// TIA Portal V19 export
DATA_BLOCK "A02_Carriage"   // DB159, Motion_DB
// stored: InstanceOfName TO_SynchronousAxis, OfSystemLibElement TO_SynchronousAxis, OfSystemLibVersion 8.0
TO_SynchronousAxis   // technology object, version 8.0
// stored: Connection Interface Actor, InputAddress 3264, OutputAddress 3264
// stored: Connection Interface Sensor[1], InputAddress 3264, OutputAddress 3264, SensorIndexInActorTelegram 1
// stored: Connection Interface Sensor[2], InputAddress 3264, OutputAddress 3264, SensorIndexInActorTelegram 2
// stored: ActualValueCoupling Ref A02_Rollformer, Type TO_PositioningAxis
   // // inherited from TO_PositioningAxis
   // // inherited from TO_SpeedAxis
   // // inherited from TO_Axis
   // // inherited from TO_Object
   // VAR
   //    Actor : TO_Struct_Actor;
   //    DynamicLimits : TO_Struct_DynamicLimits;
   //    DynamicDefaults : TO_Struct_DynamicDefaults;
   // END_VAR
   // VAR
   //    Sensor : Array[1..4] of TO_Struct_Sensor;
   //    Mechanics : TO_Struct_Mechanics;
   //    PositionLimits_HW : TO_Struct_PositionLimitsHW;
   //    Homing : TO_Struct_Homing;
   //    PositionControl : TO_Struct_PositionControl;
   //    DynamicAxisModel : TO_Struct_DynamicAxisModel;
   //    FollowingError : TO_Struct_FollowingError;
   //    StandstillSignal : TO_Struct_StandstillSignal;
   // END_VAR
   // VAR
   //    StatusSynchronizedMotion { ExternalWritable := 'False'; S7_SetPoint := 'True'} : TO_Struct_StatusSynchronizedMotion;
   // END_VAR
BEGIN
   Actor.DataAdaption := 1;
   Actor.Interface.AddressIn.RID := 16#208072c;
   Actor.Interface.AddressIn.AREA := 16#81;
   Actor.Interface.AddressIn.OFFSET := 3264;
   Actor.Interface.AddressOut.RID := 16#208072d;
   Actor.Interface.AddressOut.AREA := 16#82;
   Actor.Interface.AddressOut.OFFSET := 3264;
   Actor.DriveParameter.ReferenceSpeed := 2000.0;
   Actor.DriveParameter.MaxSpeed := 4046.462;
   Actor.DriveParameter.ReferenceTorque := 168.27;
   DynamicLimits.MaxVelocity := 50000.0;
   DynamicLimits.Velocity := 50000.0;
   DynamicLimits.MaxAcceleration := 5000.0;
   DynamicLimits.MaxDeceleration := 5000.0;
   DynamicLimits.MaxJerk := 99999.9999999997;
   DynamicDefaults.Velocity := 6000.0;
   DynamicDefaults.EmergencyDeceleration := 5000.0;
   Sensor[2].Existent := true;
   Sensor[1]."Type" := 2;
   Sensor[2].System := 0;
   Sensor[1..2].DataAdaption := 1;
   Sensor[1].ActualVelocityMode := 1;
   Sensor[1..2].Interface.AddressIn.RID := 16#208072c;
   Sensor[1..2].Interface.AddressIn.AREA := 16#81;
   Sensor[1..2].Interface.AddressIn.OFFSET := 3264;
   Sensor[1..2].Interface.AddressOut.RID := 16#208072d;
   Sensor[1..2].Interface.AddressOut.AREA := 16#82;
   Sensor[1..2].Interface.AddressOut.OFFSET := 3264;
   Sensor[2].Interface.Number := 2;
   Sensor[2].Parameter.Resolution := 0.004;
   Sensor[1].Parameter.DeterminableRevolutions := 4096;
   Sensor[1].Parameter.ReferenceSpeed := 2000.0;
   Mechanics.LeadScrew := 25.0;
   PositionLimits_HW.Active := true;
   PositionLimits_HW.MinSwitchLevel := false;
   PositionLimits_HW.MinSwitchAddress.RID := 16#2000001;
   PositionLimits_HW.MinSwitchAddress.AREA := 16#81;
   PositionLimits_HW.MinSwitchAddress.OFFSET := 2960;
   PositionLimits_HW.MaxSwitchLevel := false;
   PositionLimits_HW.MaxSwitchAddress.RID := 16#2000001;
   PositionLimits_HW.MaxSwitchAddress.AREA := 16#81;
   PositionLimits_HW.MaxSwitchAddress.OFFSET := 2961;
   PositionLimits_HW.ApproachBehavior := 1;
   Homing.ApproachVelocity := 6000.0;
   Homing.ReferencingVelocity := 1500.0;
   PositionControl.Kv := 60.0;
   PositionControl.EnableDSC := true;
   DynamicAxisModel.VelocityTimeConstant := 0.00157556176185608;
   FollowingError.MinVelocity := 600.0;
   StandstillSignal.VelocityThreshold := 300.0;
   _Units.VelocityUnit := 1524;
   Sensor[2].Existent := True;
   Sensor[2].Interface.Number := 2;
   _PositionLimits_HW.MinSwitchAddress := FlyingCarriage_MinStroke;
   _PositionLimits_HW.MaxSwitchAddress := FlyingCarriage_MaxStroke;
   _Actor.Interface.Telegram := 106;
   _Actor.DataAdaptionOffline := True;
   _Sensor[1].Interface.Telegram := 106;
   _Sensor[1].DataAdaptionOffline := True;
   _Sensor[2].Interface.Telegram := 106;
   _Sensor[2].DataAdaptionOffline := True;
END_DATA_BLOCK
